// TIA Portal V16 export
// export: Created 2023-03-29T11:03:40.2669753Z, ExportSetting WithDefaults, DisplayName Totally Integrated Automation Portal, DisplayVersion V16 Update 6, DisplayName TIA Portal Version Control Interface, DisplayVersion V16 Update 2, DisplayName TIA Portal Openness, DisplayVersion V16 Update 6, DisplayName STEP 7 Professional, DisplayVersion V16 Update 6, DisplayName STEP 7 Safety, DisplayVersion V16, DisplayName WinCC Advanced, DisplayVersion V16 Update 6
DATA_BLOCK "Nastawy_Parametrów_Sterownia_DB"   // DB69
AUTHOR : rtecmer
VERSION : 0.1
// stored: AutoNumber true, DBAccessibleFromOPCUA true, InstanceOfName Nastawy_Parametrów_Sterownia, InstanceOfType FB
"Nastawy_Parametrów_Sterownia"
BEGIN
END_DATA_BLOCK
